// TIA Portal project "tutorial tanque de agua" (V15)

(* hardware
DEVICE "S7-1200 station_1"  S7-1200 Station
   slot 0: "Rack_0"  S7-1200 Rack  Rack  V1.0
   slot 1: "PLC_1"  CPU 1214C AC/DC/Rly  6ES7 214-1BE30-0XB0  V2.2
   slot 3: "AQ 1x12BIT_1"  AQ1 signal board  6ES7 232-4HA30-0XB0  V1.0
DEVICE "S7-1200 station_2"  S7-1200 Station
   slot 0: "Rack_0"  S7-1200 Rack  Rack  V1.0
   slot 1: "PLC_2"  CPU 1214C AC/DC/Rly  6ES7 214-1BG40-0XB0  V4.2
   slot 3: "AQ 1x12BIT_1"  AQ1 signal board  6ES7 232-4HA30-0XB0  V1.0
DEVICE "HMI_2"  KTP700 Basic PN
   slot 0: "HMI_2"  KTP700 Basic PN  6AV2 123-2GB03-0AX0  15.0.0.0
   slot 1: "HMI_RT_2"  KTP700 Basic PN  6AV2 123-2GB03-0AX0  15.0.0.0
   slot 5: "HMI_2.IE_CP_1"  PROFINET Interface  15.0.0.0
      slot 1: "Interfaz PROFINET_1"  PROFINET Interface
         slot 1: "Port_1"  Port
DEVICE "HMI_1"  KTP700 Basic PN
   slot 0: "HMI_1"  KTP700 Basic PN  6AV2 123-2GB03-0AX0  15.0.0.0
   slot 1: "HMI_RT_1"  KTP700 Basic PN  6AV2 123-2GB03-0AX0  15.0.0.0
   slot 5: "HMI_1.IE_CP_1"  PROFINET Interface  15.0.0.0
      slot 1: "Interfaz PROFINET_1"  PROFINET Interface
         slot 1: "Port_1"  Port
*)

// ===== PLC "PLC_1"  CPU 1214C AC/DC/Rly =====

VAR_GLOBAL   // PLC tag table "Tabla de variables estándar"
   "H" AT %MD40 : Real;   // altura máxima del tanque
   "D" AT %MD44 : Real;   // diametro tanque
   "VOL max" AT %MD48 : Real;   // volumen maximo de llenado
   "ALTURA" AT %MD60 : Real;   // altura real de agua
   "VOLUMEN" AT %MD64 : Real;   // volumen actual
   "BIT DE ERROR" AT %Q1.7 : Bool;   // Error al realizar el cálculo
   "TENSION_real" AT %MD70 : Real;
   "ENTRADA NORM" AT %MD90 : Real;
   "VOLTAJE" AT %IW64 : Int;
   "N MULTIPLICADO" AT %MD94 : Real;
   "TENSION ESCALADA A 100" AT %MD98 : Real;
   "TENSION IMAGINARIA" AT %MD102 : Real;
   "TENSION A ESCALAR" AT %MD106 : Real;
END_VAR

FUNCTION "Cálculo de volumen de tanque" : Void   // FC140, SCL
{ S7_Optimized_Access := 'TRUE' }
VERSION : 0.1
   VAR_INPUT
      diametro : Real;
      "altura de llenado" : Real;
      "altura maxima" : Real;
   END_VAR
   VAR_OUTPUT
      volumen : Real;
      "volumen max" : Real;
      er : Bool;
   END_VAR
BEGIN
   //
   //
   IF #"altura de llenado">=0 AND #"altura de llenado"<=#"altura maxima" AND #diametro >0 THEN
       #volumen := SQR(#diametro) / 4 * 3.14159 * #"altura de llenado" * 1000;
       #"volumen max" := SQR(#diametro) / 4 * 3.14159 * #"altura maxima" * 1000;
       #er:=FALSE;
   ELSE
       #volumen := -1;
       #er:= TRUE;

   END_IF;
END_FUNCTION

ORGANIZATION_BLOCK "Main"   // OB1, LAD, ProgramCycle
TITLE = "Main Program Sweep (Cycle)"
{ S7_Optimized_Access := 'TRUE' }
VERSION : 0.1
BEGIN

REGION Network 1: Entrada de datos y cálculo de volumen
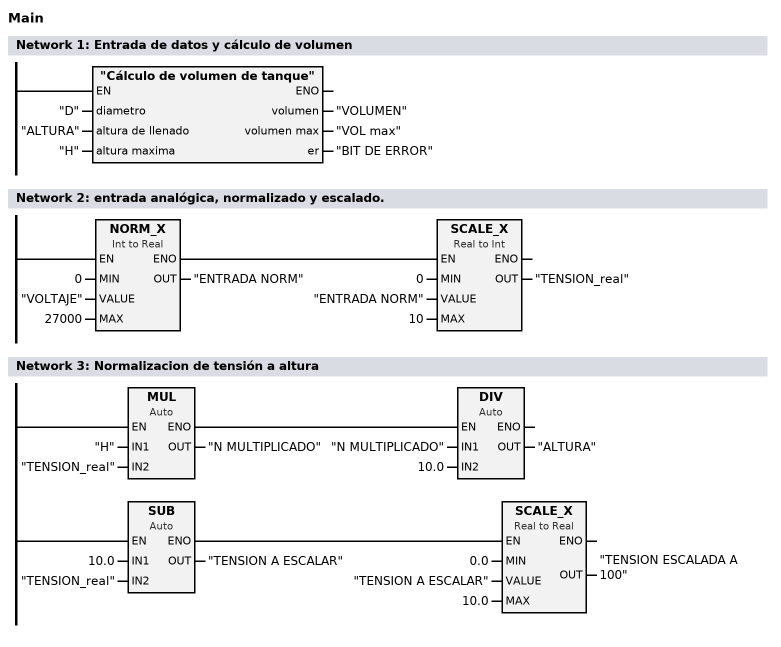
   RUNG wire#powerrail
      "Cálculo de volumen de tanque"(diametro := "D", "altura de llenado" := "ALTURA", "altura maxima" := "H", volumen => "VOLUMEN", "volumen max" => "VOL max", er => "BIT DE ERROR")
   END_RUNG
   // the same network as SCL:
   "Cálculo de volumen de tanque"(diametro := "D",
                           "altura de llenado" := "ALTURA",
                           "altura maxima" := "H",
                           volumen => "VOLUMEN",
                           "volumen max" => "VOL max",
                           er => "BIT DE ERROR");
END_REGION

REGION Network 2: entrada analógica, normalizado y escalado.
   RUNG wire#powerrail
      { S7_Templates := "[SrcType := Int, DestType := Real]"; S7_GenerateENO := "TRUE" } Normalize(min := 0, value := "VOLTAJE", max := 27000, out => "ENTRADA NORM")
      { S7_Templates := "[SrcType := Real, DestType := Int]"; S7_GenerateENO := "TRUE" } Scale(min := 0, value := "ENTRADA NORM", max := 10, out => "TENSION_real")
   END_RUNG
   // the same network as SCL:
   // ENO of a box is taken as its EN; it also drops when the box reports an error
   "ENTRADA NORM" := NORM_X(MIN := 0, VALUE := "VOLTAJE", MAX := 27000);
   "TENSION_real" := SCALE_X(MIN := 0, VALUE := "ENTRADA NORM", MAX := 10);
END_REGION

REGION Network 3: Normalizacion de tensión a altura
   RUNG wire#powerrail
      { S7_GenerateENO := "TRUE" } Mul(in1 := "H", in2 := "TENSION_real", out => "N MULTIPLICADO")
      { S7_GenerateENO := "TRUE" } Div(in1 := "N MULTIPLICADO", in2 := 10.0, out => "ALTURA")
   END_RUNG
   RUNG wire#powerrail
      { S7_GenerateENO := "TRUE" } Sub(in1 := 10.0, in2 := "TENSION_real", out => "TENSION A ESCALAR")
      { S7_Templates := "[SrcType := Real, DestType := Real]"; S7_GenerateENO := "TRUE" } Scale(min := 0.0, value := "TENSION A ESCALAR", max := 10.0, out => "TENSION ESCALADA A 100")
   END_RUNG
   // the same network as SCL:
   // ENO of a box is taken as its EN; it also drops when the box reports an error
   "N MULTIPLICADO" := "H" * "TENSION_real";
   "ALTURA" := "N MULTIPLICADO" / 10.0;
   "TENSION A ESCALAR" := 10.0 - "TENSION_real";
   "TENSION ESCALADA A 100" := SCALE_X(MIN := 0.0, VALUE := "TENSION A ESCALAR", MAX := 10.0);
END_REGION
END_ORGANIZATION_BLOCK

// ===== PLC "PLC_2"  CPU 1214C AC/DC/Rly =====

VAR_GLOBAL   // PLC tag table "Tabla de variables estándar"
   "H" AT %MD40 : Real;   // altura máxima del tanque
   "D" AT %MD44 : Real;   // diametro tanque
   "VOL max" AT %MD48 : Real;   // volumen maximo de llenado
   "ALTURA" AT %MD60 : Real;   // altura real de agua
   "VOLUMEN" AT %MD64 : Real;   // volumen actual
   "BIT DE ERROR" AT %Q1.7 : Bool;   // Error al realizar el cálculo
   "TENSION_real" AT %MD70 : Real;
   "ENTRADA NORM" AT %MD90 : Real;
   "VOLTAJE" AT %IW64 : Int;
   "N MULTIPLICADO" AT %MD94 : Real;
   "TENSION ESCALADA A 100" AT %MD98 : Real;
   "TENSION IMAGINARIA" AT %MD102 : Real;
END_VAR

FUNCTION "Cálculo de volumen de tanque" : Void   // FC140, SCL
{ S7_Optimized_Access := 'TRUE' }
VERSION : 0.1
   VAR_INPUT
      diametro : Real;
      "altura de llenado" : Real;
      "altura maxima" : Real;
   END_VAR
   VAR_OUTPUT
      volumen : Real;
      "volumen max" : Real;
      er : Bool;
   END_VAR
BEGIN
   //
   //
   IF #"altura de llenado">=0 AND #"altura de llenado"<=#"altura maxima" AND #diametro >0 THEN
       #volumen := SQR(#diametro) / 4 * 3.14159 * #"altura de llenado" * 1000;
       #"volumen max" := SQR(#diametro) / 4 * 3.14159 * #"altura maxima" * 1000;
       #er:=FALSE;
   ELSE
       #volumen := -1;
       #er:= TRUE;

   END_IF;
END_FUNCTION

ORGANIZATION_BLOCK "Main"   // OB1, LAD, ProgramCycle
TITLE = "Main Program Sweep (Cycle)"
{ S7_Optimized_Access := 'TRUE' }
VERSION : 0.1
   VAR_INPUT
      Initial_Call : Bool;   // Initial call of this OB
      Remanence : Bool;   // =True, if remanent data are available
   END_VAR
BEGIN

REGION Network 1
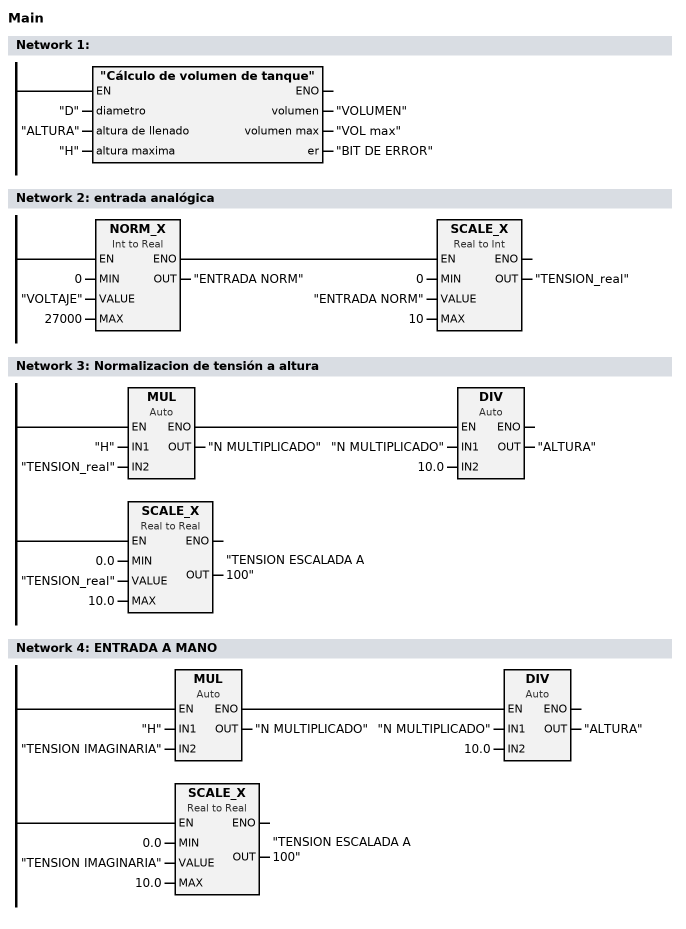
   RUNG wire#powerrail
      "Cálculo de volumen de tanque"(diametro := "D", "altura de llenado" := "ALTURA", "altura maxima" := "H", volumen => "VOLUMEN", "volumen max" => "VOL max", er => "BIT DE ERROR")
   END_RUNG
   // the same network as SCL:
   "Cálculo de volumen de tanque"(diametro := "D",
                           "altura de llenado" := "ALTURA",
                           "altura maxima" := "H",
                           volumen => "VOLUMEN",
                           "volumen max" => "VOL max",
                           er => "BIT DE ERROR");
END_REGION

REGION Network 2: entrada analógica
   RUNG wire#powerrail
      { S7_Templates := "[SrcType := Int, DestType := Real]"; S7_GenerateENO := "TRUE" } Normalize(min := 0, value := "VOLTAJE", max := 27000, out => "ENTRADA NORM")
      { S7_Templates := "[SrcType := Real, DestType := Int]"; S7_GenerateENO := "TRUE" } Scale(min := 0, value := "ENTRADA NORM", max := 10, out => "TENSION_real")
   END_RUNG
   // the same network as SCL:
   // ENO of a box is taken as its EN; it also drops when the box reports an error
   "ENTRADA NORM" := NORM_X(MIN := 0, VALUE := "VOLTAJE", MAX := 27000);
   "TENSION_real" := SCALE_X(MIN := 0, VALUE := "ENTRADA NORM", MAX := 10);
END_REGION

REGION Network 3: Normalizacion de tensión a altura
   RUNG wire#powerrail
      Mul(in1 := "H", in2 := "TENSION_real", out => "N MULTIPLICADO")
      Div(in1 := "N MULTIPLICADO", in2 := 10.0, out => "ALTURA")
   END_RUNG
   RUNG wire#powerrail
      { S7_Templates := "[SrcType := Real, DestType := Real]" } Scale(min := 0.0, value := "TENSION_real", max := 10.0, out => "TENSION ESCALADA A 100")
   END_RUNG
   // the same network as SCL:
   "N MULTIPLICADO" := "H" * "TENSION_real";
   "ALTURA" := "N MULTIPLICADO" / 10.0;
   "TENSION ESCALADA A 100" := SCALE_X(MIN := 0.0, VALUE := "TENSION_real", MAX := 10.0);
END_REGION

REGION Network 4: ENTRADA A MANO
   RUNG wire#powerrail
      Mul(in1 := "H", in2 := "TENSION IMAGINARIA", out => "N MULTIPLICADO")
      Div(in1 := "N MULTIPLICADO", in2 := 10.0, out => "ALTURA")
   END_RUNG
   RUNG wire#powerrail
      { S7_Templates := "[SrcType := Real, DestType := Real]" } Scale(min := 0.0, value := "TENSION IMAGINARIA", max := 10.0, out => "TENSION ESCALADA A 100")
   END_RUNG
   // the same network as SCL:
   "N MULTIPLICADO" := "H" * "TENSION IMAGINARIA";
   "ALTURA" := "N MULTIPLICADO" / 10.0;
   "TENSION ESCALADA A 100" := SCALE_X(MIN := 0.0, VALUE := "TENSION IMAGINARIA", MAX := 10.0);
END_REGION
END_ORGANIZATION_BLOCK

(* ===== HMI "HMI_RT_2" =====
system functions are stored by id; their names below are inferred from use
connection "HMI_Conexión_2": ETHERNET, SMART_S7_1200_OMS

HMI tags "Tabla de variables estándar"
   "Número_imagen_variable" : UInt, internal
   "H" : Real = PLC H AT %MD40, 1 s
   "D" : Real = PLC D AT %MD44, 1 s
   "ALTURA" : Real = PLC ALTURA AT %MD60, 1 s
   "VOLUMEN" : Real = PLC VOLUMEN AT %MD64, 1 s
   "VOL max" : Real = PLC "VOL max" AT %MD48, 1 s
   "TENSION ESCALADA A 100" : Real = PLC "TENSION ESCALADA A 100" AT %MD98, 1 s
   "ENTRADA NORM" : Real = PLC "ENTRADA NORM" AT %MD90, 1 s
   "TENSION_real" : Real = PLC TENSION_real AT %MD70, 1 s
   "VOLTAJE" : Int = PLC VOLTAJE AT %IW64, 1 s
   "TENSION IMAGINARIA" : Real = PLC "TENSION IMAGINARIA" AT %MD102, 1 s

text list "Nombre_imagen_lista_texto": 1 'Imagen raíz'

Template "Plantilla_1" 800x480
   Button "Salir" at 714,429 size 71x50; TextOff 'Salir'; PictureOff "ExitRuntime_KTP700_Basic_PN_TR"; PictureOn "ExitRuntime_KTP700_Basic_PN_TR"
      on Release: StopRuntime(0)
   Button "Template_Button" at 614,429 size 71x50; TextOff 'Text'
   Button "Template_Button_1" at 514,429 size 71x50; TextOff 'Text'
   Button "Template_Button_2" at 414,429 size 71x50; TextOff 'Text'
   Button "Template_Button_3" at 314,429 size 71x50; TextOff 'Text'
   Button "Template_Button_4" at 214,429 size 71x50; TextOff 'Text'
   Button "Avisos" at 114,429 size 71x50; TextOff 'Avisos'; PictureOff "AlarmDisplay_KTP700_Basic_PN_TR"; PictureOn "AlarmDisplay_KTP700_Basic_PN_TR"
      on Release: function_ef3f5d25("Ventana de avisos_no_acusado", -1)
   Button "Imagen inicial" at 14,429 size 71x50; TextOff 'Imagen inicial'; PictureOff "NavigateHome_KTP700_Basic_PN_TR"; PictureOn "NavigateHome_KTP700_Basic_PN_TR"
      on Release: ActivateScreen("Imagen raíz", 0)
   SymbolicIOField "Imagen_campo_ES_simbólico" at 93,9 size 600x33; TextOff '0'; TextOn '1'; TextList "Nombre_imagen_lista_texto"
      ProcessValue <- "Número_imagen_variable"
      on Change: ActivateScreenByNumber("Número_imagen_variable", 0)
   DateTimeField "HmiScreenItemData" at 695,25 size 105x25
   DateTimeField "HmiScreenItemData_1" at 695,0 size 105x25
   GraphicView "Logotipo" at 0,0 size 91x51; Picture "Logotipo de HMI_2"

screen "Imagen raíz" 800x480, template "Plantilla_1"
   on GenerateScreen: SetTag("Número_imagen_variable", 1)
   Bar "Barra_1" at 257,148 size 246x283; MinimumValue 0; MaximumValue 100
      ProcessValue <- "TENSION ESCALADA A 100"
   IOField "Campo ES_1" at 33,116 size 96x32; FormatPattern s999999999.999
      ProcessValue <- "H"
   IOField "Campo ES_2" at 34,242 size 96x32; FormatPattern s999999999.999
      ProcessValue <- "D"
   IOField "Campo ES_4" at 609,174 size 96x32; FormatPattern s999999999.999
      ProcessValue <- "VOLUMEN"
   IOField "Campo ES_5" at 609,316 size 96x32; FormatPattern s999999999.999
      ProcessValue <- "VOL max"
   IOField "Campo ES_3" at 33,357 size 96x32; FormatPattern s999999999.999
      ProcessValue <- "TENSION IMAGINARIA"
   TextField "Campo de texto_1" at 34,88 size 115x23; Text 'ALTURA MAX'
   TextField "Campo de texto_2" at 34,213 size 95x23; Text 'DIÁMETRO'
   TextField "Campo de texto_3" at 34,334 size 79x23; Text 'TENSION'
   TextField "Campo de texto_4" at 605,144 size 85x23; Text 'VOLUMEN'
   TextField "Campo de texto_5" at 604,290 size 127x23; Text 'VOLUMEN MAX'
*)

(* ===== HMI "HMI_RT_1" =====
system functions are stored by id; their names below are inferred from use
connection "HMI_Conexión_1": ETHERNET, SMART_S7_1200_OMS

HMI tags "Tabla de variables estándar"
   "Número_imagen_variable" : UInt, internal
   "TENSION ESCALADA A 100" : Real = PLC "TENSION ESCALADA A 100" AT %MD98, 100 ms
   "H" : Real = PLC H AT %MD40, 1 s
   "D" : Real = PLC D AT %MD44, 1 s
   "VOLUMEN" : Real = PLC VOLUMEN AT %MD64, 100 ms
   "VOL max" : Real = PLC "VOL max" AT %MD48, 1 s

text list "Nombre_imagen_lista_texto": 1 'Imagen raíz'

Template "Plantilla_1" 800x480
   Button "Salir" at 714,429 size 71x50; TextOff 'Salir'; PictureOff "ExitRuntime_KTP700_Basic_PN_TR"; PictureOn "ExitRuntime_KTP700_Basic_PN_TR"
      on Release: StopRuntime(0)
   Button "Template_Button" at 614,429 size 71x50; TextOff 'Text'
   Button "Template_Button_1" at 514,429 size 71x50; TextOff 'Text'
   Button "Template_Button_2" at 414,429 size 71x50; TextOff 'Text'
   Button "Template_Button_3" at 314,429 size 71x50; TextOff 'Text'
   Button "Template_Button_4" at 214,429 size 71x50; TextOff 'Text'
   Button "Avisos" at 114,429 size 71x50; TextOff 'Avisos'; PictureOff "AlarmDisplay_KTP700_Basic_PN_TR"; PictureOn "AlarmDisplay_KTP700_Basic_PN_TR"
      on Release: function_ef3f5d25("Ventana de avisos_no_acusado", -1)
   Button "Imagen inicial" at 14,429 size 71x50; TextOff 'Imagen inicial'; PictureOff "NavigateHome_KTP700_Basic_PN_TR"; PictureOn "NavigateHome_KTP700_Basic_PN_TR"
      on Release: ActivateScreen("Imagen raíz", 0)
   SymbolicIOField "Imagen_campo_ES_simbólico" at 93,9 size 600x33; TextOff '0'; TextOn '1'; TextList "Nombre_imagen_lista_texto"
      ProcessValue <- "Número_imagen_variable"
      on Change: ActivateScreenByNumber("Número_imagen_variable", 0)
   DateTimeField "HmiScreenItemData" at 695,25 size 105x25
   DateTimeField "HmiScreenItemData_1" at 695,0 size 105x25
   GraphicView "Logotipo" at 0,0 size 91x51; Picture "Logotipo de HMI_1"

screen "Imagen raíz" 800x480, template "Plantilla_1"
   on GenerateScreen: SetTag("Número_imagen_variable", 1)
   Bar "Barra_1" at 301,101 size 195x245; MinimumValue 0; MaximumValue 100
      ProcessValue <- "TENSION ESCALADA A 100"
   IOField "Campo ES_1" at 81,127 size 96x32; FormatPattern s999999999.999
      ProcessValue <- "H"
   IOField "Campo ES_2" at 81,239 size 96x32; FormatPattern s999999999.999
      ProcessValue <- "D"
   IOField "Campo ES_3" at 587,148 size 96x32; FormatPattern s999999999.999
      ProcessValue <- "VOLUMEN"
   IOField "Campo ES_4" at 587,255 size 96x32; FormatPattern s999999999.999
      ProcessValue <- "VOL max"
   TextField "Campo de texto_1" at 81,82 size 115x23; Text 'ALTURA MAX'
   TextField "Campo de texto_2" at 82,206 size 95x23; Text 'DIAMETRO'
   TextField "Campo de texto_3" at 586,109 size 85x23; Text 'VOLUMEN'
   TextField "Campo de texto_4" at 587,221 size 160x23; Text 'VOLUMEN MAXIMO'
*)